// TIA Portal V19 export
FUNCTION "ChainWash" : Void   // FC97, STL
TITLE = CHAIN WASH
{ S7_Optimized_Access := 'TRUE' }
NAME : CIPTANK
VERSION : 0.0
// Comment
// stored: AutoNumber false
BEGIN

NETWORK
TITLE = CHAIN WASH
// Comment
      AN    "S0 CHAIN WASH";
      R     "S1 CHAIN WASH";
      R     "S2 CHAIN WASH";
      R     "S3 CHAIN WASH";
      BEC;

//    Step 1 Set route chain wash
      A     "S1 CHAIN WASH";
      JC    M001;
      R     "MM0139";
      R     "MY0114";  // drain
      S     "MY0116";
      S     "MY0117";
      R     "MY0119";
      R     "AutoTT0172/IP0157";
      R     "ManTT0172/IP0157";
      S     "S1 CHAIN WASH";
      BEU;
M001: NOP   0;

NETWORK
TITLE = 
// Comment  Step 2 Wait for route to be ready
      A     "S2 CHAIN WASH";
      JC    c001;
      AN    "Y0116S";
      BEC;
      AN    "Y0117S";
      BEC;
      S     "S2 CHAIN WASH";
      BEU;
c001: NOP   0;

NETWORK
TITLE = Prerinse
// Comment  Step 3 Wait for "CHIAN WASH" signal from filler machine
      A     "S3 CHAIN WASH";
      JC    c002;
      AN    "CHAIN_WASH";
      BEC;
      S     "CONTROL CIP TANK";
      S     "MY0115";
      S     "S3 CHAIN WASH";
      BEU;
c002: NOP   0;

NETWORK
TITLE = Prerinse
// Comment  Step 4 Wait for level in balance tank 01.40
      AN    "B01.42";
      R     "AutoTT0172/IP0157";
      R     "MY0158";
      BEC;
      L     "Setpoints".ChainWashTempSetp;  // "DB SETPOINTS".ChainWashTempSetp
      T     "PID_TT0172/IP0157".TT0172SpDBD;
      S     "AutoTT0172/IP0157";
      S     "MY0158";
      S     "MM0139";
      BEU;

END_FUNCTION
